// TIA Portal V19 export
DATA_BLOCK "MwFakCalc_PS"   // DB211
{ S7_Optimized_Access := 'TRUE' }
// stored: MemoryReserve 100
   VAR
      StartMeasure { S7_SetPoint := 'True'} : Bool;
      AuxStartMeasure : Bool;
      MeasureID : UInt;
      MeasuredValueG : LReal;
      MeasuredValueW : LReal;
   END_VAR
BEGIN
END_DATA_BLOCK
